SYSTEM test
  (* Version 1.0, 2022-12-03, hf *)
  APPLICATION App1
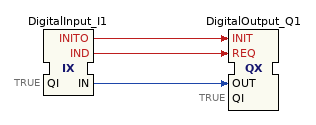
    FBS
      DigitalInput_I1 : IX(QI := TRUE);
      DigitalOutput_Q1 : QX(QI := TRUE);
    END_FBS
    EVENT_CONNECTIONS
      DigitalInput_I1.INITO TO DigitalOutput_Q1.INIT;
      DigitalInput_I1.IND TO DigitalOutput_Q1.REQ;
    END_CONNECTIONS
    DATA_CONNECTIONS
      DigitalInput_I1.IN TO DigitalOutput_Q1.OUT;
    END_CONNECTIONS
  END_APPLICATION
  APPLICATION Mapping
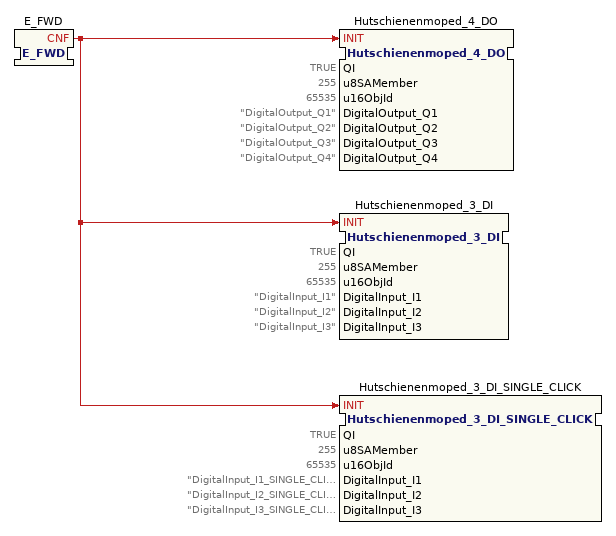
    FBS
      Hutschienenmoped_3_DI : Hutschienenmoped_3_DI(QI := TRUE, u8SAMember := 255, u16ObjId := 65535, DigitalInput_I1 := "DigitalInput_I1", DigitalInput_I2 := "DigitalInput_I2", DigitalInput_I3 := "DigitalInput_I3");
      Hutschienenmoped_3_DI_SINGLE_CLICK : Hutschienenmoped_3_DI_SINGLE_CLICK(QI := TRUE, u8SAMember := 255, u16ObjId := 65535, DigitalInput_I1 := "DigitalInput_I1_SINGLE_CLICK", DigitalInput_I2 := "DigitalInput_I2_SINGLE_CLICK", DigitalInput_I3 := "DigitalInput_I3_SINGLE_CLICK");
      E_FWD : E_FWD;
      Hutschienenmoped_4_DO : Hutschienenmoped_4_DO(QI := TRUE, u8SAMember := 255, u16ObjId := 65535, DigitalOutput_Q1 := "DigitalOutput_Q1", DigitalOutput_Q2 := "DigitalOutput_Q2", DigitalOutput_Q3 := "DigitalOutput_Q3", DigitalOutput_Q4 := "DigitalOutput_Q4");
    END_FBS
    EVENT_CONNECTIONS
      E_FWD.CNF TO Hutschienenmoped_3_DI.INIT;
      E_FWD.CNF TO Hutschienenmoped_3_DI_SINGLE_CLICK.INIT;
      E_FWD.CNF TO Hutschienenmoped_4_DO.INIT;
    END_CONNECTIONS
  END_APPLICATION
  APPLICATION App2
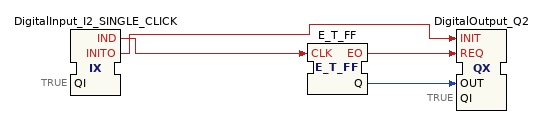
    FBS
      E_T_FF : E_T_FF;
      DigitalInput_I2_SINGLE_CLICK : IX(QI := TRUE);
      DigitalOutput_Q2 : QX(QI := TRUE);
    END_FBS
    EVENT_CONNECTIONS
      DigitalInput_I2_SINGLE_CLICK.IND TO E_T_FF.CLK;
      DigitalInput_I2_SINGLE_CLICK.INITO TO DigitalOutput_Q2.INIT;
      E_T_FF.EO TO DigitalOutput_Q2.REQ;
    END_CONNECTIONS
    DATA_CONNECTIONS
      E_T_FF.Q TO DigitalOutput_Q2.OUT;
    END_CONNECTIONS
  END_APPLICATION
  DEVICE FORTE_PC : FORTE_PC(MGR_ID := "localhost:61499")
    {SET_ATTRIBUTE(Profile, HOLOBLOC)}
    RESOURCE EMB_RES : EMB_RES
      FBS
        E_FWD : E_FWD;
        Hutschienenmoped_3_DI_SINGLE_CLICK : Hutschienenmoped_3_DI_SINGLE_CLICK(QI := TRUE, u8SAMember := 255, u16ObjId := 65535, DigitalInput_I1 := "DigitalInput_I1_SINGLE_CLICK", DigitalInput_I2 := "DigitalInput_I2_SINGLE_CLICK", DigitalInput_I3 := "DigitalInput_I3_SINGLE_CLICK");
        Hutschienenmoped_3_DI : Hutschienenmoped_3_DI(QI := TRUE, u8SAMember := 255, u16ObjId := 65535, DigitalInput_I1 := "DigitalInput_I1", DigitalInput_I2 := "DigitalInput_I2", DigitalInput_I3 := "DigitalInput_I3");
        Hutschienenmoped_4_DO : Hutschienenmoped_4_DO(QI := TRUE, u8SAMember := 255, u16ObjId := 65535, DigitalOutput_Q1 := "DigitalOutput_Q1", DigitalOutput_Q2 := "DigitalOutput_Q2", DigitalOutput_Q3 := "DigitalOutput_Q3", DigitalOutput_Q4 := "DigitalOutput_Q4");
        E_T_FF : E_T_FF;
        DigitalInput_I1 : IX(QI := TRUE);
        DigitalInput_I2_SINGLE_CLICK : IX(QI := TRUE);
        DigitalOutput_Q1 : QX(QI := TRUE);
        DigitalOutput_Q2 : QX(QI := TRUE);
      END_FBS
      EVENT_CONNECTIONS
        E_FWD.CNF TO Hutschienenmoped_3_DI_SINGLE_CLICK.INIT;
        E_FWD.CNF TO Hutschienenmoped_3_DI.INIT;
        E_FWD.CNF TO Hutschienenmoped_4_DO.INIT;
        DigitalInput_I2_SINGLE_CLICK.IND TO E_T_FF.CLK;
        DigitalInput_I1.INITO TO DigitalOutput_Q1.INIT;
        DigitalInput_I1.IND TO DigitalOutput_Q1.REQ;
        DigitalInput_I2_SINGLE_CLICK.INITO TO DigitalOutput_Q2.INIT;
        E_T_FF.EO TO DigitalOutput_Q2.REQ;
      END_CONNECTIONS
      DATA_CONNECTIONS
        DigitalInput_I1.IN TO DigitalOutput_Q1.OUT;
        E_T_FF.Q TO DigitalOutput_Q2.OUT;
      END_CONNECTIONS
    END_RESOURCE
  END_DEVICE
  MAPPINGS
    Mapping.E_FWD ON FORTE_PC.EMB_RES.E_FWD;
    Mapping.Hutschienenmoped_3_DI_SINGLE_CLICK ON FORTE_PC.EMB_RES.Hutschienenmoped_3_DI_SINGLE_CLICK;
    Mapping.Hutschienenmoped_3_DI ON FORTE_PC.EMB_RES.Hutschienenmoped_3_DI;
    Mapping.Hutschienenmoped_4_DO ON FORTE_PC.EMB_RES.Hutschienenmoped_4_DO;
    App2.E_T_FF ON FORTE_PC.EMB_RES.E_T_FF;
    App1.DigitalInput_I1 ON FORTE_PC.EMB_RES.DigitalInput_I1;
    App2.DigitalInput_I2_SINGLE_CLICK ON FORTE_PC.EMB_RES.DigitalInput_I2_SINGLE_CLICK;
    App1.DigitalOutput_Q1 ON FORTE_PC.EMB_RES.DigitalOutput_Q1;
    App2.DigitalOutput_Q2 ON FORTE_PC.EMB_RES.DigitalOutput_Q2;
  END_MAPPINGS
  SEGMENTS
    Ethernet : Ethernet;
  END_SEGMENTS
  LINKS
    FORTE_PC => Ethernet;
  END_LINKS
END_SYSTEM
